TYPE E_TURN_DIRECTION :
(
	AUTOMATIC := 0,
	LEFT := 1,
	RIGHT := 2,
	MAX_E_TURN_DIRECTION
);
END_TYPE

(* stored: Version 1.1.0.1, ProductVersion 3.1.0.26
   DUT E_TURN_DIRECTION: Id {c64f9134-9c1a-4730-886a-ba6e51a4143f} *)
